// TwinCAT 3 PLC project Untitled1
// ProgramVersion: 3.1.4023.0
// libraries:
//   Tc2_MC2, * (Beckhoff Automation GmbH)
//   Tc2_Standard, * (Beckhoff Automation GmbH)
//   Tc2_System, * (Beckhoff Automation GmbH)
//   Tc2_Utilities, * (Beckhoff Automation GmbH)
//   Tc3_Module, * (Beckhoff Automation GmbH)
// project tree:
//   DUTs/Motion Package/Drives/ AirPiston.TcPOU (not stored), ClearLinkMC.TcPOU (not stored), ServoNC.TcPOU, CenteredServoNC.TcPOU, SimplePiston.TcPOU (not stored)
//   DUTs/Motion Package/ Homing.TcDUT (not stored), Insertion.TcPOU (not stored), SuctionPad.TcDUT (not stored)
//   DUTs/Motion Package/Prototypes/ FBA_Drive.TcPOU (not stored), FBA_TrifectaDrive.TcPOU (not stored), I_ContinuousDrive.TcIO (not stored), I_Drive.TcIO (not stored), I_EncodedDrive.TcIO (not stored), I_PositionalDrive.TcIO (not stored)
//   DUTs/Robots/ KukaRobot.TcPOU, RobotA26.TcPOU (not stored), TaskA26.TcDUT
//   DUTs/ SectionEnum.TcDUT (not stored), Watchdog.TcPOU (not stored)
//   / PlcTask.TcTTO
//   POUs/ DataIsEmpty.TcPOU (not stored), MAIN.TcPOU, SpacerRecollectionUnit.TcPOU
// real-time tasks:
//   TASK PlcTask: cycle T#10ms, priority 20, ADS port 350

CONFIGURATION Untitled1
    RESOURCE PLC ON TwinCAT3
        TASK PlcTask(INTERVAL := T#10ms, PRIORITY := 20);
        PROGRAM MAIN WITH PlcTask : MAIN;
    END_RESOURCE
END_CONFIGURATION

// ---- DUTs/Robots/TaskA26.TcDUT
{attribute 'qualified_only'}
{attribute 'to_string'}
TYPE TaskA26 :
(
	IDLE,
	PICK_SPACER,
	
	size
);
END_TYPE

// ---- POUs/MAIN.TcPOU
PROGRAM MAIN
VAR_OUTPUT
	localTime : TIMESTRUCT; //used by watchdogs, not set in module
END_VAR
VAR
	spacerRecollector : SpacerRecollectionUnit;
END_VAR
VAR
	robot7 : RobotA26;
	robotSliderA26 : ServoNC := (
		limitSensorDefaultState := TRUE,
		enableDualSideTraverse := TRUE);
		
END_VAR
VAR //sensors to detect spacers on receiver conveyors
	spacerPresent_A24_LRC_C02 AT %I* : BOOL;
	spacerPresent_A24_LRC_C04 AT %I* : BOOL;
	spacerPresent_A24_LRC_C06 AT %I* : BOOL;
	spacerPresent_A24_LRC_C08 AT %I* : BOOL;
	spacerPresent_A24_LRC_C10 AT %I* : BOOL;
	spacerPresent_A24_LRC_C12 AT %I* : BOOL;
END_VAR

CallHardware(); //start program with hardware call
SetupHardware(); //not applicable for this module

runModules();

CallHardware(); //end program with hardware call

METHOD PROTECTED callHardware : BOOL
VAR_INPUT
END_VAR
robot7(bEnable:= TRUE, abort:= , conveyorSafety:= TRUE);	
robotSliderA26(bEnable:= TRUE, ready=> , position=> , velocity=> );
END_METHOD

METHOD PROTECTED runModules : BOOL
VAR_INPUT
END_VAR
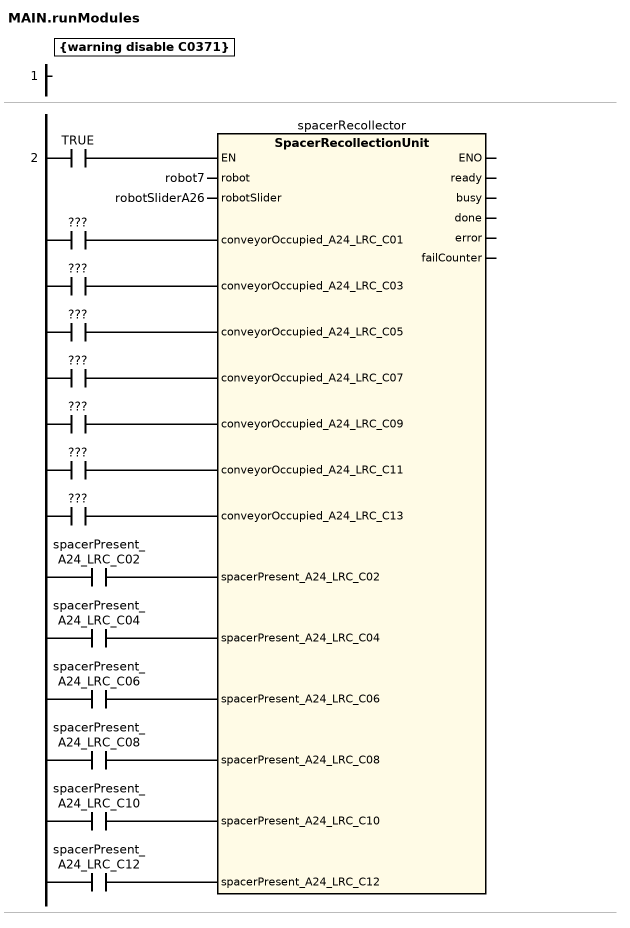
// NETWORK 1
// label: {warning disable C0371}

// NETWORK 2
spacerRecollector(
    robot := robot7,
    robotSlider := robotSliderA26,
    spacerPresent_A24_LRC_C02 := spacerPresent_A24_LRC_C02,
    spacerPresent_A24_LRC_C04 := spacerPresent_A24_LRC_C04,
    spacerPresent_A24_LRC_C06 := spacerPresent_A24_LRC_C06,
    spacerPresent_A24_LRC_C08 := spacerPresent_A24_LRC_C08,
    spacerPresent_A24_LRC_C10 := spacerPresent_A24_LRC_C10,
    spacerPresent_A24_LRC_C12 := spacerPresent_A24_LRC_C12); // SpacerRecollectionUnit
END_METHOD

METHOD PROTECTED setupHardware : BOOL
VAR
	
END_VAR
END_METHOD

END_PROGRAM

// ---- POUs/SpacerRecollectionUnit.TcPOU
FUNCTION_BLOCK SpacerRecollectionUnit //EXTENDS SectionEx
VAR_IN_OUT
	robot : RobotA26;
	robotSlider : ServoNC;
END_VAR
VAR_INPUT
	conveyorOccupied_A24_LRC_C01 : BOOL;
	conveyorOccupied_A24_LRC_C03 : BOOL;
	conveyorOccupied_A24_LRC_C05 : BOOL;
	conveyorOccupied_A24_LRC_C07 : BOOL;
	conveyorOccupied_A24_LRC_C09 : BOOL;
	conveyorOccupied_A24_LRC_C11 : BOOL;
	conveyorOccupied_A24_LRC_C13 : BOOL;
	
	spacerPresent_A24_LRC_C02 : BOOL;
	spacerPresent_A24_LRC_C04 : BOOL;
	spacerPresent_A24_LRC_C06 : BOOL;
	spacerPresent_A24_LRC_C08 : BOOL;
	spacerPresent_A24_LRC_C10 : BOOL;
	spacerPresent_A24_LRC_C12 : BOOL;
END_VAR
VAR_OUTPUT
	ready : BOOL;
	busy : BOOL;
	done : BOOL;
	error : BOOL;
	
	failCounter : INT;
END_VAR
VAR
	step : (IDLE, SLIDE, PICK_SPACER, COMPLETE);
	iPosition : INT;
END_VAR
VAR //slider positions
	pickPos1, pickPos2 : LREAL;
END_VAR

ready := step = 0;
busy := step > 0;
done := done;
error := error;

IF 
	conveyorOccupied_A24_LRC_C01 OR
	conveyorOccupied_A24_LRC_C03 OR
	conveyorOccupied_A24_LRC_C05 OR
	conveyorOccupied_A24_LRC_C07 OR
	conveyorOccupied_A24_LRC_C09 OR
	conveyorOccupied_A24_LRC_C11 OR
	conveyorOccupied_A24_LRC_C13
THEN
	robot.clearCommand();
	
ELSE
	//remove spacers from transfer conveyors in ascending order
	process();
	
END_IF

METHOD process : BOOL
VAR
	spacersPresent : ARRAY[1..6] OF BOOL := [
		spacerPresent_A24_LRC_C02,
		spacerPresent_A24_LRC_C04,
		spacerPresent_A24_LRC_C06,
		spacerPresent_A24_LRC_C08,
		spacerPresent_A24_LRC_C10,
		spacerPresent_A24_LRC_C12];
END_VAR
VAR CONSTANT
	suctionDistance : INT := 10;
END_VAR
{warning disable C0371}

iPosition := MAX(1, iPosition); //value is always at least 1

CASE step OF
	IDLE:
		IF DataIsEmpty(arr := ADR(spacersPresent), arrSize := SIZEOF(spacersPresent)) THEN
			robotSlider.toHome();
			
			iPosition := 0;
			failCounter := 0;
			process := TRUE;
		
		ELSIF NOT spacersPresent[iPosition] THEN
			iPosition := iPosition + 1;
			
		ELSIF robot.Ready THEN
			step := SLIDE;
		END_IF
		
	SLIDE:
		CASE iPosition OF
			1,2,3:		robotSlider.moveAbsolute(newTarget := pickPos1);
			4,5,6:		robotSlider.moveAbsolute(newTarget := pickPos2);
		END_CASE
		
		//replace this condition with WithinTolerance() if the slider spends too long adjusting its position
		IF robotSlider.CurrentPosition = robotSlider.TargetPosition THEN
			step := PICK_SPACER;
		END_IF
		
	PICK_SPACER:		
		IF robot.eoatDistance > suctionDistance THEN
			robot.HoldMaterial := 'SPACER';
		ELSE
			robot.HoldMaterial := '';
		END_IF
	
		IF robot.Done THEN
			step := COMPLETE;
		ELSE
			robot.setGroup(group := 1, value := TaskA26.PICK_SPACER);
			robot.setGroup(group := 2, value := iPosition);
		END_IF
		
	COMPLETE:
		robot.HoldMaterial := '';
		
		IF spacersPresent[iPosition] THEN
			failCounter := failCounter + 1;
		END_IF
		
		robot.clearCommand();
		step := 0;
	
END_CASE
END_METHOD

END_FUNCTION_BLOCK

// ---- DUTs/Motion Package/Drives/ServoNC.TcPOU
FUNCTION_BLOCK ServoNC EXTENDS FBA_TrifectaDrive IMPLEMENTS I_EncodedDrive
VAR_OUTPUT	
	ready : BOOL;
	position : LREAL;
	velocity : LREAL;
END_VAR
VAR
	axis : AXIS_REF;
	
	mcReadPosition : MC_ReadActualPosition; //continuous enable FBs
	mcReadVelocity : MC_ReadActualVelocity;
	mcReadError : MC_ReadAxisError;
	mcPower : MC_Power;
	
	mcReset : MC_Reset; //rising edge FBs
	mcMoveAbsolute : MC_MoveAbsolute;
	mcMoveRelative : MC_MoveRelative;
	mcMoveVelocity : MC_MoveVelocity;
	
	mcSetPosition : MC_SetPosition;
	mcStop : MC_Stop;
END_VAR
VAR_STAT CONSTANT
	targetingVelocity : INT := 500;
	continuousVelocity : INT := 100;
END_VAR

override();

blocks();

mcReset.Execute := FALSE;
mcMoveAbsolute.Execute := FALSE;
mcMoveRelative.Execute := FALSE;
mcMoveVelocity.Execute := FALSE;
mcSetPosition.Execute := FALSE;
mcStop.Execute := FALSE;

blocks();

ready := bEnable AND NOT Active AND HomeSet;

PROPERTY Active : BOOL
GET
Active := 
	mcMoveAbsolute.Busy OR 
	mcMoveRelative.Busy OR 
	mcMoveVelocity.Busy OR 
	mcSetPosition.Busy OR 
	mcReset.Busy OR 
	mcStop.Busy OR 
	step <> 0;
END_GET
END_PROPERTY

METHOD PRIVATE blocks : BOOL
mcReadPosition(
	Axis:= axis, 
	Enable:= TRUE, 
	Valid=> , 
	Busy=> , 
	Error=> , 
	ErrorID=> , 
	Position=> position);
	
mcReadVelocity(
	Axis:= axis, 
	Enable:= TRUE, 
	Valid=> , 
	Busy=> , 
	Error=> , 
	ErrorID=> , 
	ActualVelocity=> velocity);
	
mcReadError(
	Axis:= axis, 
	Enable:= TRUE, 
	Valid=> , 
	Busy=> , 
	Error=> , 
	ErrorID=> , 
	AxisErrorID=> );

mcReset(
	Axis:= axis, 
	Execute:= , 
	Done=> , 
	Busy=> , 
	Error=> , 
	ErrorID=> );

mcPower(
	Axis:= axis, 
	Enable:= bEnable, 
	Enable_Positive:= TRUE, 
	Enable_Negative:= TRUE, 
	Override:= 100, 
	BufferMode:= , 
	Options:= , 
	Status=> , 
	Busy=> , 
	Active=> , 
	Error=> , 
	ErrorID=> );

mcMoveAbsolute(
	Axis:= axis, 
	Execute:= , 
	Position:= , 
	Velocity:= targetingVelocity, 
	Acceleration:= , 
	Deceleration:= , 
	Jerk:= , 
	BufferMode:= , 
	Options:= , 
	Done=> , 
	Busy=> , 
	Active=> , 
	CommandAborted=> , 
	Error=> , 
	ErrorID=> );
	
mcMoveRelative(
	Axis:= axis, 
	Execute:= , 
	Distance:= ,
	Velocity:= targetingVelocity, 
	Acceleration:= , 
	Deceleration:= , 
	Jerk:= , 
	BufferMode:= , 
	Options:= , 
	Done=> , 
	Busy=> , 
	Active=> , 
	CommandAborted=> , 
	Error=> , 
	ErrorID=> );
	
mcMoveVelocity( //stopped with stop();
	Axis:= axis, 
	Execute:= , 
	Velocity:= continuousVelocity, 
	Acceleration:= , 
	Deceleration:= , 
	Jerk:= , 
	Direction:= , 
	BufferMode:= , 
	Options:= , 
	InVelocity=> , 
	Busy=> , 
	Active=> , 
	CommandAborted=> , 
	Error=> , 
	ErrorID=> );
	
mcSetPosition(
	Axis:= axis, 
	Execute:= , 
	Position:= , 
	Mode:= , 
	Options:= , 
	Done=> , 
	Busy=> , 
	Error=> , 
	ErrorID=> );
	
mcStop(
	Axis:= axis, 
	Execute:= , 
	Deceleration:= , 
	Jerk:= , 
	Options:= , 
	Done=> , 
	Busy=> , 
	Active=> , 
	CommandAborted=> , 
	Error=> , 
	ErrorID=> );
END_METHOD

PROPERTY CurrentPosition : LREAL
GET
CurrentPosition := position;
END_GET
SET
position := CurrentPosition;
END_SET
END_PROPERTY

PROPERTY Error : BOOL
GET
error := 
	mcMoveAbsolute.Error OR 
	mcMoveRelative.Error OR 
	mcMoveVelocity.Error OR 
	mcSetPosition.Error OR 
	mcReset.Error OR 
	mcStop.Error OR
	mcReadError.AxisErrorID > 0;
END_GET
END_PROPERTY

METHOD homingSequence : BOOL
CASE step OF
	Homing.IDLE:
		reset();
		IF bEnable THEN
			step := Homing.START;
		END_IF
		
	Homing.START:
		IF AtHome THEN
			mcMoveVelocity.Execute := FALSE;
			step := Homing.STOP;
			
		ELSIF AtInnerLimit THEN
			mcMoveVelocity.Execute := FALSE;
			step := Homing.RETRY;
			
		ELSE
			mcMoveVelocity.Direction := MC_Negative_Direction;
			mcMoveVelocity.Execute := NOT mcMoveVelocity.Execute;
		END_IF
		
	Homing.RETRY:
		IF AtOuterLimit THEN
			mcMoveVelocity.Execute := FALSE;
			step := Homing.START;
		ELSE
			mcMoveVelocity.Direction := MC_Positive_Direction;
			mcMoveVelocity.Execute := NOT mcMoveVelocity.Execute;
		END_IF
		
	Homing.STOP:
		IF velocity = 0 THEN
			mcStop.Execute := FALSE;
			step := Homing.SET;
		ELSE
			mcStop.Execute := TRUE;
		END_IF
		
	Homing.SET:
		IF position = 0 THEN
			mcSetPosition.Execute := FALSE;
			homingSequence := TRUE;
			step := Homing.DONE;
		ELSE
			mcSetPosition.Position := 0;
			mcSetPosition.Execute := TRUE;
		END_IF
		
	Homing.DONE:
		homingComplete := TRUE;
		step := Homing.IDLE;
		
END_CASE
END_METHOD

METHOD moveAbsolute : BOOL
VAR_INPUT
	newTarget : LREAL;
END_VAR
(*
VAR_OUTPUT
	fault : BOOL;
END_VAR
*)
IF NOT Active AND NOT error THEN
	mcMoveAbsolute.Position := newTarget;
	mcMoveAbsolute.Execute := TRUE;
END_IF

moveAbsolute := (*mcMoveAbsolute.Done AND mcMoveAbsolute.Active;*)
	position = newTarget;
END_METHOD

METHOD moveContinuous : BOOL
VAR_INPUT
	//direction : BOOL; //direction (F = inwards, T = outwards)
	direction : MC_Direction;
END_VAR
(*
IF mcMoveVelocity.Active THEN
	stop();
END_IF

IF NOT mcStop.Done THEN
	RETURN;
END_IF
*)
(*
IF direction THEN
	mcMoveVelocity.Direction := MC_Positive_Direction;
ELSE
	mcMoveVelocity.Direction := MC_Negative_Direction;
END_IF
*)
mcMoveVelocity.Direction := direction;

IF NOT mcMoveVelocity.Error THEN
	mcMoveVelocity.Execute := TRUE;
	moveContinuous := TRUE;
END_IF
END_METHOD

METHOD moveRelative : BOOL
VAR_INPUT
	distance : LREAL;
END_VAR
mcMoveRelative.Distance := distance;

moveRelative := mcMoveRelative.Done;
END_METHOD

METHOD PRIVATE override : BOOL
VAR_INPUT
END_VAR
(*
-at home and attempting to traverse outward
-at outer limit and attempting to traverse outward
-at inner limit and attempting to traverse inwards
*)
(*
inward = negative direction, negative velocity
outward = positive direction, positive velocity
*)

IF error THEN
	stop();
	reset();
	
ELSIF
	(NOT enableDualSideTraverse AND AtHome AND (TargetPosition > CurrentPosition OR velocity > 0)) OR
	(AtInnerLimit AND (TargetPosition > CurrentPosition OR velocity > 0)) OR
	(AtOuterLimit AND (TargetPosition < CurrentPosition OR velocity < 0))
THEN
	stop();
END_IF

//if enableTraversePastHome, then first condition is ignored
END_METHOD

METHOD reset : BOOL
VAR_INPUT
END_VAR
mcReset.Execute := TRUE;

reset := mcReset.Done;
END_METHOD

METHOD stop : BOOL
VAR_INPUT
END_VAR
mcStop.Execute := TRUE;

mcMoveAbsolute.Execute := FALSE;
mcMoveRelative.Execute := FALSE;
mcMoveVelocity.Execute := FALSE;
END_METHOD

PROPERTY TargetPosition : LREAL
GET
END_GET
SET
moveAbsolute(newTarget := TargetPosition);
END_SET
END_PROPERTY

METHOD toHome : BOOL
VAR_INPUT
END_VAR
moveAbsolute(newTarget := 0);

toHome := AtHome;
END_METHOD

END_FUNCTION_BLOCK

// ---- DUTs/Motion Package/Drives/CenteredServoNC.TcPOU
FUNCTION_BLOCK CenteredServoNC EXTENDS FBA_TrifectaDrive IMPLEMENTS I_EncodedDrive
VAR_OUTPUT	
	ready : BOOL;
	position : LREAL;
	velocity : LREAL;
END_VAR
VAR
	axis : AXIS_REF;
	
	mcReadPosition : MC_ReadActualPosition; //continuous enable FBs
	mcReadVelocity : MC_ReadActualVelocity;
	mcReadError : MC_ReadAxisError;
	mcPower : MC_Power;
	
	mcReset : MC_Reset; //rising edge FBs
	mcMoveAbsolute : MC_MoveAbsolute;
	mcMoveRelative : MC_MoveRelative;
	mcMoveVelocity : MC_MoveVelocity;
	
	mcSetPosition : MC_SetPosition;
	mcStop : MC_Stop;
END_VAR
VAR_STAT CONSTANT
	targetingVelocity : INT := 500;
	continuousVelocity : INT := 100;
END_VAR

(*
NOTE:
	this servo is almost identical to ServoNC, only difference being this servo can travel to both left and right limits
	the entire motion control heirarchy is messy and needs reworking
*)

override();

blocks();

mcReset.Execute := FALSE;
mcMoveAbsolute.Execute := FALSE;
mcMoveRelative.Execute := FALSE;
mcMoveVelocity.Execute := FALSE;
mcSetPosition.Execute := FALSE;
mcStop.Execute := FALSE;

blocks();

ready := bEnable AND NOT Active AND HomeSet;

PROPERTY Active : BOOL
GET
Active := 
	mcMoveAbsolute.Busy OR 
	mcMoveRelative.Busy OR 
	mcMoveVelocity.Busy OR 
	mcSetPosition.Busy OR 
	mcReset.Busy OR 
	mcStop.Busy OR 
	step <> 0;
END_GET
END_PROPERTY

METHOD PRIVATE blocks : BOOL
mcReadPosition(
	Axis:= axis, 
	Enable:= TRUE, 
	Valid=> , 
	Busy=> , 
	Error=> , 
	ErrorID=> , 
	Position=> position);
	
mcReadVelocity(
	Axis:= axis, 
	Enable:= TRUE, 
	Valid=> , 
	Busy=> , 
	Error=> , 
	ErrorID=> , 
	ActualVelocity=> velocity);
	
mcReadError(
	Axis:= axis, 
	Enable:= TRUE, 
	Valid=> , 
	Busy=> , 
	Error=> , 
	ErrorID=> , 
	AxisErrorID=> );

mcReset(
	Axis:= axis, 
	Execute:= , 
	Done=> , 
	Busy=> , 
	Error=> , 
	ErrorID=> );

mcPower(
	Axis:= axis, 
	Enable:= bEnable, 
	Enable_Positive:= TRUE, 
	Enable_Negative:= TRUE, 
	Override:= 100, 
	BufferMode:= , 
	Options:= , 
	Status=> , 
	Busy=> , 
	Active=> , 
	Error=> , 
	ErrorID=> );

mcMoveAbsolute(
	Axis:= axis, 
	Execute:= , 
	Position:= , 
	Velocity:= targetingVelocity, 
	Acceleration:= , 
	Deceleration:= , 
	Jerk:= , 
	BufferMode:= , 
	Options:= , 
	Done=> , 
	Busy=> , 
	Active=> , 
	CommandAborted=> , 
	Error=> , 
	ErrorID=> );
	
mcMoveRelative(
	Axis:= axis, 
	Execute:= , 
	Distance:= ,
	Velocity:= targetingVelocity, 
	Acceleration:= , 
	Deceleration:= , 
	Jerk:= , 
	BufferMode:= , 
	Options:= , 
	Done=> , 
	Busy=> , 
	Active=> , 
	CommandAborted=> , 
	Error=> , 
	ErrorID=> );
	
mcMoveVelocity( //stopped with stop();
	Axis:= axis, 
	Execute:= , 
	Velocity:= continuousVelocity, 
	Acceleration:= , 
	Deceleration:= , 
	Jerk:= , 
	Direction:= , 
	BufferMode:= , 
	Options:= , 
	InVelocity=> , 
	Busy=> , 
	Active=> , 
	CommandAborted=> , 
	Error=> , 
	ErrorID=> );
	
mcSetPosition(
	Axis:= axis, 
	Execute:= , 
	Position:= , 
	Mode:= , 
	Options:= , 
	Done=> , 
	Busy=> , 
	Error=> , 
	ErrorID=> );
	
mcStop(
	Axis:= axis, 
	Execute:= , 
	Deceleration:= , 
	Jerk:= , 
	Options:= , 
	Done=> , 
	Busy=> , 
	Active=> , 
	CommandAborted=> , 
	Error=> , 
	ErrorID=> );
END_METHOD

PROPERTY CurrentPosition : LREAL
GET
CurrentPosition := position;
END_GET
SET
position := CurrentPosition;
END_SET
END_PROPERTY

PROPERTY Error : BOOL
GET
error := 
	mcMoveAbsolute.Error OR 
	mcMoveRelative.Error OR 
	mcMoveVelocity.Error OR 
	mcSetPosition.Error OR 
	mcReset.Error OR 
	mcStop.Error OR
	mcReadError.AxisErrorID > 0;
END_GET
END_PROPERTY

METHOD homingSequence : BOOL
CASE step OF
	Homing.IDLE:
		reset();
		IF bEnable THEN
			step := Homing.START;
		END_IF
		
	Homing.START:
		IF AtHome THEN
			mcMoveVelocity.Execute := FALSE;
			step := Homing.STOP;
			
		ELSIF AtInnerLimit THEN
			mcMoveVelocity.Execute := FALSE;
			step := Homing.RETRY;
			
		ELSE
			mcMoveVelocity.Direction := MC_Negative_Direction;
			mcMoveVelocity.Execute := NOT mcMoveVelocity.Execute;
		END_IF
		
	Homing.RETRY:
		IF AtOuterLimit THEN
			mcMoveVelocity.Execute := FALSE;
			step := Homing.START;
		ELSE
			mcMoveVelocity.Direction := MC_Positive_Direction;
			mcMoveVelocity.Execute := NOT mcMoveVelocity.Execute;
		END_IF
		
	Homing.STOP:
		IF velocity = 0 THEN
			mcStop.Execute := FALSE;
			step := Homing.SET;
		ELSE
			mcStop.Execute := TRUE;
		END_IF
		
	Homing.SET:
		IF position = 0 THEN
			mcSetPosition.Execute := FALSE;
			homingSequence := TRUE;
			step := Homing.DONE;
		ELSE
			mcSetPosition.Position := 0;
			mcSetPosition.Execute := TRUE;
		END_IF
		
	Homing.DONE:
		homingComplete := TRUE;
		step := Homing.IDLE;
		
END_CASE
END_METHOD

METHOD moveAbsolute : BOOL
VAR_INPUT
	newTarget : LREAL;
END_VAR
(*
VAR_OUTPUT
	fault : BOOL;
END_VAR
*)
IF NOT Active AND NOT error THEN
	mcMoveAbsolute.Position := newTarget;
	mcMoveAbsolute.Execute := TRUE;
END_IF

moveAbsolute := (*mcMoveAbsolute.Done AND mcMoveAbsolute.Active;*)
	position = newTarget;
END_METHOD

METHOD moveContinuous : BOOL
VAR_INPUT
	//direction : BOOL; //direction (F = inwards, T = outwards)
	direction : MC_Direction;
END_VAR
(*
IF mcMoveVelocity.Active THEN
	stop();
END_IF

IF NOT mcStop.Done THEN
	RETURN;
END_IF
*)
(*
IF direction THEN
	mcMoveVelocity.Direction := MC_Positive_Direction;
ELSE
	mcMoveVelocity.Direction := MC_Negative_Direction;
END_IF
*)
mcMoveVelocity.Direction := direction;

IF NOT mcMoveVelocity.Error THEN
	mcMoveVelocity.Execute := TRUE;
	moveContinuous := TRUE;
END_IF
END_METHOD

METHOD moveRelative : BOOL
VAR_INPUT
	distance : LREAL;
END_VAR
mcMoveRelative.Distance := distance;

moveRelative := mcMoveRelative.Done;
END_METHOD

METHOD PRIVATE override : BOOL
VAR_INPUT
END_VAR
(*
-at home and attempting to traverse outward
-at outer limit and attempting to traverse outward
-at inner limit and attempting to traverse inwards
*)
(*
inward = negative direction, negative velocity
outward = positive direction, positive velocity
*)

IF error THEN
	stop();
	reset();
	
ELSIF
	//AtHome AND (TargetPosition > CurrentPosition OR velocity > 0) OR //condition removed, servo can traverse on either side of home
	AtInnerLimit AND (TargetPosition > CurrentPosition OR velocity > 0) OR
	AtOuterLimit AND (TargetPosition < CurrentPosition OR velocity < 0)
THEN
	stop();
END_IF
END_METHOD

METHOD reset : BOOL
VAR_INPUT
END_VAR
mcReset.Execute := TRUE;

reset := mcReset.Done;
END_METHOD

METHOD stop : BOOL
VAR_INPUT
END_VAR
mcStop.Execute := TRUE;

mcMoveAbsolute.Execute := FALSE;
mcMoveRelative.Execute := FALSE;
mcMoveVelocity.Execute := FALSE;
END_METHOD

PROPERTY TargetPosition : LREAL
GET
END_GET
SET
moveAbsolute(newTarget := TargetPosition);
END_SET
END_PROPERTY

METHOD toHome : BOOL
VAR_INPUT
END_VAR
moveAbsolute(newTarget := 0);

toHome := AtHome;
END_METHOD

END_FUNCTION_BLOCK

// ---- DUTs/Robots/KukaRobot.TcPOU
FUNCTION_BLOCK KukaRobot
VAR_INPUT
	bEnable : BOOL := TRUE; //this enables the robot
	abort : BOOL := FALSE; //this disables the robot
	//bEnable must be TRUE and abort must be FALSE for the robot to function
END_VAR
VAR_OUTPUT
	(*
	forceStop AT %Q* : BOOL;
	resetSignal AT %Q* : BOOL;
	*)
	
	reservation : INT := 0;
	
	error : BOOL;
	errId : DINT;
	
	outputs AT %Q* : ARRAY[1..20] OF WORD;
	inputs AT %I* : ARRAY[1..20] OF WORD;
END_VAR
VAR
	heartbeat : Watchdog;
	
	toggleBit AT %I* : BOOL; //check connection from PLC to bridge
	disconnected AT %I* : BOOL; //check connection from bridge to robot
	
	hmiReservation : STRING;
END_VAR
(*
generic KUKA robot with 20 WORD outputs and 20 WORD inputs, connected to Beckhoff IPC via EL6692 or EL6695 EtherCAT bridge
includes minimal diagnostics to detect if robot is offline
robots should always be reserved before sending a task
*)

heartbeat(
	enable:= NOT disconnected,
	toggleBit:= toggleBit,
	timeoutWidth:= T#200MS,
	timeout=> );

error := //add any addition conditions with OR
	disconnected OR
	heartbeat.timeout;
	
IF (*NOT bEnable OR*) abort THEN //bEnable is not used for now, but abort is
	stop();
END_IF

//{attribute 'monitoring' := 'variable'}
{attribute 'monitoring' := 'call'}
PROPERTY Busy : BOOL
GET
END_GET
END_PROPERTY

METHOD clearCommand : BOOL
VAR_INPUT
END_VAR
MEMSET(ADR(outputs), 0, SIZEOF(outputs));
END_METHOD

//{attribute 'monitoring' := 'variable'}
{attribute 'monitoring' := 'call'}
PROPERTY Done : BOOL
GET
END_GET
END_PROPERTY

{attribute 'monitoring' := 'call'}
PROPERTY Ready : BOOL
GET
END_GET
END_PROPERTY

METHOD release : BOOL
VAR_INPUT
	sectionReservation : INT;
END_VAR
IF reservation = sectionReservation THEN
	reservation := 0;
	release := TRUE;
END_IF
END_METHOD

METHOD reserve : BOOL
VAR_INPUT
	reserveRequest : INT;
END_VAR
(*
this method exists because chipboard and wood bunk operations use the same robot
both sections need to check if the robot is open to commands before use
*)
IF Reserved AND reservation = reserveRequest THEN
	reserve := TRUE;

ELSIF NOT Reserved THEN
	reservation := reserveRequest;
	reserve := TRUE;

END_IF
END_METHOD

{attribute 'monitoring' := 'call'}
PROPERTY Reserved : BOOL
GET
Reserved := reservation <> SectionEnum.NULL_SECTION;
END_GET
END_PROPERTY

METHOD reset : BOOL
//resetSignal := TRUE;
//done := FALSE;

MEMSET(ADR(outputs), 0, SIZEOF(outputs));
(*
IF ready AND completedTask = 0 THEN
	resetSignal := FALSE;
	reset := TRUE;
END_IF
*)
END_METHOD

METHOD resume : BOOL
VAR_INPUT
END_VAR
//forceStop := FALSE;

resume := NOT error AND errId = 0;
END_METHOD

METHOD setGroup : BOOL
VAR_INPUT
	group : INT;
	value : INT;
END_VAR
{warning disable C0195}
outputs[group] := value;
END_METHOD

METHOD stop : BOOL
VAR_INPUT
END_VAR
//forceStop := TRUE;
clearCommand();

stop := TRUE;
END_METHOD

END_FUNCTION_BLOCK
